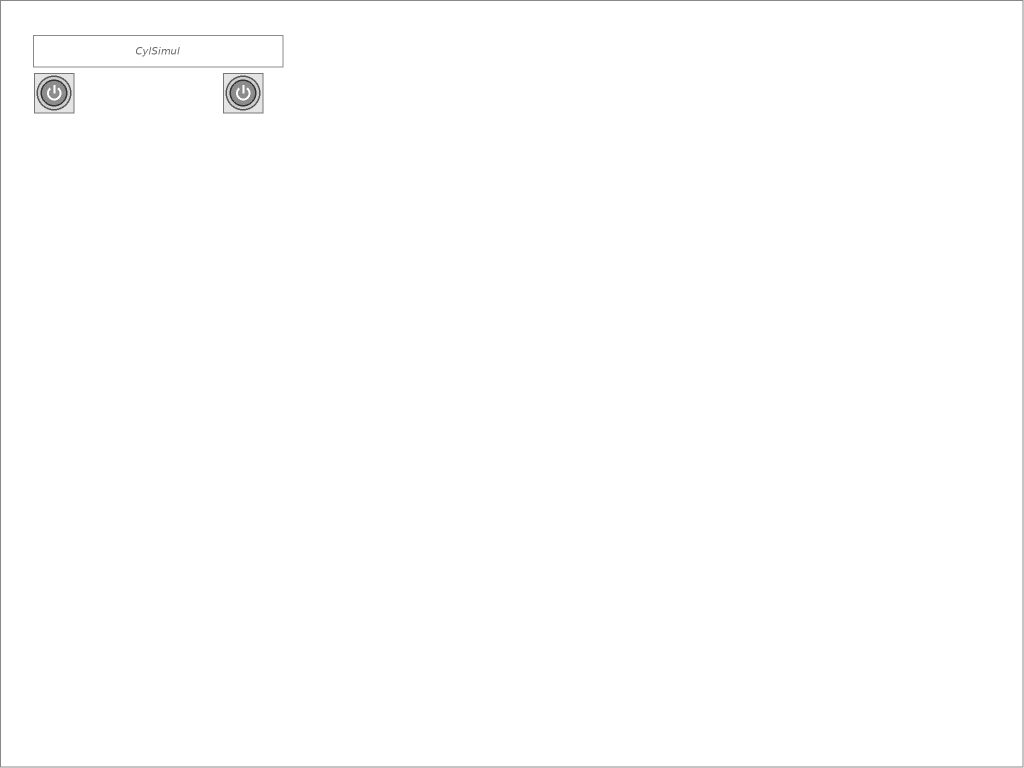
VISUALIZATION Visualization  // 1024x768
    Frame (33,35 250x32)
        shows CylSimul(currPosPercent := MAIN.offSet, sensorFwd := MAIN.sensorFwd, sensorBwd := MAIN.sensorBwd)
    PowerSwitch (34,73 40x40), variable: MAIN.recua, behaviour: TAP, style: Switch-PowerSwitch-Gray
    PowerSwitch (223,73 40x40), variable: MAIN.avanca, behaviour: TAP, style: Switch-PowerSwitch-Gray
END_VISUALIZATION

(* stored: Version 1.1.0.1, ProductVersion 3.1.4024.12
   Visu Visualization: Id {7d0c306d-2fd1-4518-99c9-3a95ad3b5bdf} *)
